Staubli VAL3: fRobot2sRobot.pgx

program fRobot2sRobot()
begin

  //没有ClearBuffer 这个比较难联通

  clearBuffer(synServer)
  //把客户端收到不为空的信息通过服务器传送出去
  while true
    //服务器

    call ServerGet(sFirstRStatus)

    //call ServerSend(toString("",nPlaceCycleNum))
    delay(0)
  endWhile

end
